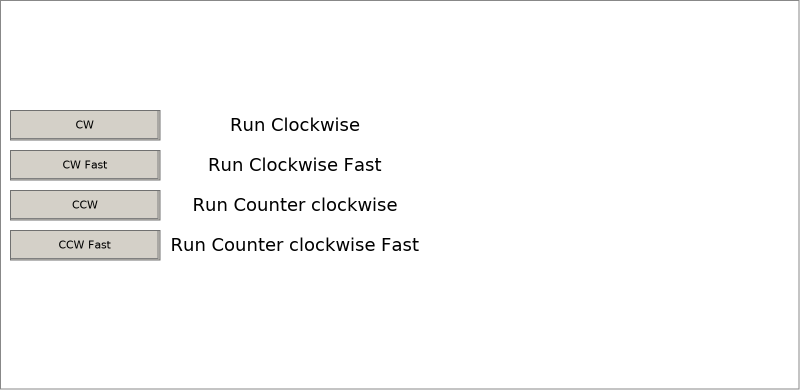
VISUALIZATION VisuTwoVelocityAxisControl  // 800x390
VAR_IN_OUT
	pDev : POINTER TO FB_DevTwoVelocityAxis;
END_VAR
    Button (10,110 150x30), "CW"
        tap pDev^.stManualControl.bManRunCW
    Button (10,150 150x30), "CW Fast"
        tap pDev^.stManualControl.bManRunCWFast
    Button (10,190 150x30), "CCW"
        tap pDev^.stManualControl.bManRunCCw
    Button (10,230 150x30), "CCW Fast"
        tap pDev^.stManualControl.bManRunCCWFast
    Label (170,110 250x30), "Run Clockwise"
    Label (170,150 250x30), "Run Clockwise Fast"
    Label (170,190 250x30), "Run Counter clockwise"
    Label (170,230 250x30), "Run Counter clockwise Fast"
END_VISUALIZATION

(* stored: Version 1.1.0.1, ProductVersion 3.1.4024.11
   Visu VisuTwoVelocityAxisControl: Id {d68122d0-aa3c-06f4-2457-39f06616d4fb} *)
